// TIA Portal project "Project19" (V15.1)

(* hardware
DEVICE "S7-1200 station_1"  S7-1200 Station
   slot 0: "Rack_0"  S7-1200 Rack  Rack  V1.0
   slot 1: "PLC_1"  CPU 1214C DC/DC/DC  6ES7 214-1AG40-0XB0  V4.2
*)

// ===== PLC "PLC_1"  CPU 1214C DC/DC/DC =====

VAR_GLOBAL   // PLC tag table "Default tag table"
   "BE" AT %I0.0 : Bool;
   "LIGA" AT %I0.1 : Bool;
   "DESLIGA" AT %I0.2 : Bool;
   "SA0" AT %I0.3 : Bool;
   "SA1" AT %I0.4 : Bool;
   "SB0" AT %I0.5 : Bool;
   "SB1" AT %I0.6 : Bool;
   "SC0" AT %I0.7 : Bool;
   "SC1" AT %I1.0 : Bool;
   "SD0" AT %I1.1 : Bool;
   "SD1" AT %I1.2 : Bool;
   "AVANÇA A" AT %Q0.1 : Bool;
   "AVANÇA B" AT %Q0.2 : Bool;
   "AVANÇA C" AT %Q0.3 : Bool;
   "AVANÇA D" AT %Q0.4 : Bool;
   "RECUA A" AT %Q0.5 : Bool;
   "RECUA B" AT %Q0.6 : Bool;
   "RECUA C" AT %Q0.7 : Bool;
   "RECUA D" AT %Q1.0 : Bool;
   "LIGADA" AT %Q1.1 : Bool;
   "FALHA" AT %Q1.2 : Bool;
   "M1" AT %M0.0 : Bool;
   "M2" AT %M0.1 : Bool;
   "M3" AT %M0.2 : Bool;
   "M4" AT %M0.3 : Bool;
   "M5" AT %M0.4 : Bool;
   "M6" AT %M0.5 : Bool;
   "M7" AT %M0.6 : Bool;
END_VAR

DATA_BLOCK "CILINDRO_A_DB"   // DB1
{ S7_Optimized_Access := 'TRUE' }
VERSION : 0.1
// stored: InstanceOfName CILINDRO
"CILINDRO"
BEGIN
END_DATA_BLOCK

DATA_BLOCK "CILINDRO_B_DB"   // DB2
{ S7_Optimized_Access := 'TRUE' }
VERSION : 0.1
// stored: InstanceOfName CILINDRO
"CILINDRO"
BEGIN
END_DATA_BLOCK

DATA_BLOCK "CILINDRO_C_DB"   // DB5
{ S7_Optimized_Access := 'TRUE' }
VERSION : 0.1
// stored: InstanceOfName CILINDRO
"CILINDRO"
BEGIN
END_DATA_BLOCK

DATA_BLOCK "CILINDRO_D_DB"   // DB7
{ S7_Optimized_Access := 'TRUE' }
VERSION : 0.1
// stored: InstanceOfName CILINDRO
"CILINDRO"
BEGIN
END_DATA_BLOCK

// folder: System blocks/Program resources

DATA_BLOCK "T1"   // DB3
{ S7_Optimized_Access := 'TRUE' }
AUTHOR : Simatic
FAMILY : IEC
NAME : IEC_TMR
VERSION : 1.0
// stored: InstanceOfName IEC_TIMER
"IEC_TIMER"
BEGIN
END_DATA_BLOCK

DATA_BLOCK "T2"   // DB4
{ S7_Optimized_Access := 'TRUE' }
AUTHOR : Simatic
FAMILY : IEC
NAME : IEC_TMR
VERSION : 1.0
// stored: InstanceOfName IEC_TIMER
"IEC_TIMER"
BEGIN
END_DATA_BLOCK

DATA_BLOCK "T3"   // DB6
{ S7_Optimized_Access := 'TRUE' }
AUTHOR : Simatic
FAMILY : IEC
NAME : IEC_TMR
VERSION : 1.0
// stored: InstanceOfName IEC_TIMER
"IEC_TIMER"
BEGIN
END_DATA_BLOCK

DATA_BLOCK "T4"   // DB8
{ S7_Optimized_Access := 'TRUE' }
AUTHOR : Simatic
FAMILY : IEC
NAME : IEC_TMR
VERSION : 1.0
// stored: InstanceOfName IEC_TIMER
"IEC_TIMER"
BEGIN
END_DATA_BLOCK

// folder: (top level)

FUNCTION_BLOCK "CILINDRO"   // FB1, LAD
{ S7_Optimized_Access := 'TRUE' }
VERSION : 0.1
   VAR_INPUT
      "COMANDO AVANÇO" : Bool;
      "COMANDO RECUO" : Bool;
      "SENSOR AVANÇO" : Bool;
      "SENSOR RECUO" : Bool;
   END_VAR
   VAR_OUTPUT
      AVANÇO : Bool;
      RECUO : Bool;
   END_VAR
BEGIN

REGION Network 1
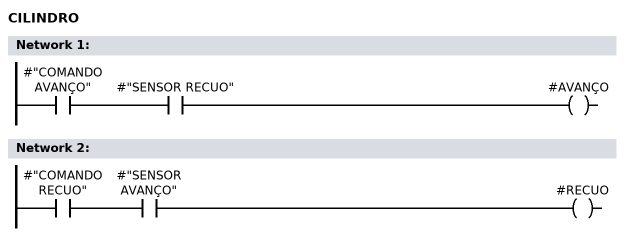
   RUNG wire#powerrail
      Contact( #"COMANDO AVANÇO" )
      Contact( #"SENSOR RECUO" )
      Coil( #AVANÇO )
   END_RUNG
   // the same network as SCL:
   #AVANÇO := #"COMANDO AVANÇO" AND #"SENSOR RECUO";
END_REGION

REGION Network 2
   RUNG wire#powerrail
      Contact( #"COMANDO RECUO" )
      Contact( #"SENSOR AVANÇO" )
      Coil( #RECUO )
   END_RUNG
   // the same network as SCL:
   #RECUO := #"COMANDO RECUO" AND #"SENSOR AVANÇO";
END_REGION
END_FUNCTION_BLOCK

FUNCTION "LOGICA DE ACIONAMENTO" : Void   // FC1, LAD
TITLE = Sequência dos cilindros
{ S7_Optimized_Access := 'TRUE' }
VERSION : 0.1
// A+B+5sA-5sB-C+5sD+5s(C-D-)
BEGIN

REGION Network 1: Selo ligado com memoria
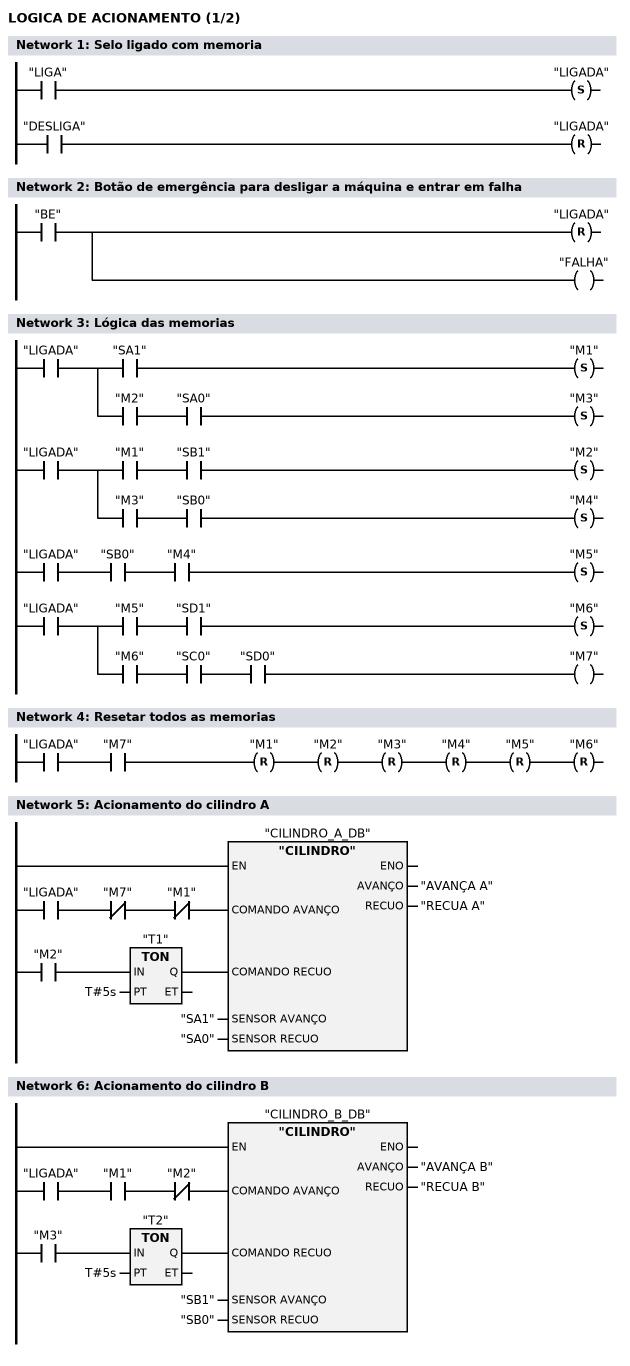
   RUNG wire#powerrail
      Contact( "LIGA" )
      S_Coil( "LIGADA" )
   END_RUNG
   RUNG wire#powerrail
      Contact( "DESLIGA" )
      R_Coil( "LIGADA" )
   END_RUNG
   // the same network as SCL:
   IF "LIGA" THEN "LIGADA" := TRUE; END_IF;
   IF "DESLIGA" THEN "LIGADA" := FALSE; END_IF;
END_REGION

REGION Network 2: Botão de emergência para desligar a máquina e entrar em falha
   RUNG wire#powerrail
      Contact( "BE" )
      wire#w1
      R_Coil( "LIGADA" )
   END_RUNG
   RUNG wire#w1
      Coil( "FALHA" )
   END_RUNG
   // the same network as SCL:
   IF "BE" THEN "LIGADA" := FALSE; END_IF;
   "FALHA" := "BE";
END_REGION

REGION Network 3: Lógica das memorias
   RUNG wire#powerrail
      Contact( "LIGADA" )
      wire#w1
      Contact( "SA1" )
      S_Coil( "M1" )
   END_RUNG
   RUNG wire#w1
      Contact( "M2" )
      Contact( "SA0" )
      S_Coil( "M3" )
   END_RUNG
   RUNG wire#powerrail
      Contact( "LIGADA" )
      wire#w2
      Contact( "M1" )
      Contact( "SB1" )
      S_Coil( "M2" )
   END_RUNG
   RUNG wire#w2
      Contact( "M3" )
      Contact( "SB0" )
      S_Coil( "M4" )
   END_RUNG
   RUNG wire#powerrail
      Contact( "LIGADA" )
      Contact( "SB0" )
      Contact( "M4" )
      S_Coil( "M5" )
   END_RUNG
   RUNG wire#powerrail
      Contact( "LIGADA" )
      wire#w3
      Contact( "M5" )
      Contact( "SD1" )
      S_Coil( "M6" )
   END_RUNG
   RUNG wire#w3
      Contact( "M6" )
      Contact( "SC0" )
      Contact( "SD0" )
      Coil( "M7" )
   END_RUNG
   // the same network as SCL:
   IF "LIGADA" AND "SA1" THEN "M1" := TRUE; END_IF;
   IF "LIGADA" AND "M2" AND "SA0" THEN "M3" := TRUE; END_IF;
   IF "LIGADA" AND "M1" AND "SB1" THEN "M2" := TRUE; END_IF;
   IF "LIGADA" AND "M3" AND "SB0" THEN "M4" := TRUE; END_IF;
   IF "LIGADA" AND "SB0" AND "M4" THEN "M5" := TRUE; END_IF;
   IF "LIGADA" AND "M5" AND "SD1" THEN "M6" := TRUE; END_IF;
   "M7" := "LIGADA" AND "M6" AND "SC0" AND "SD0";
END_REGION

REGION Network 4: Resetar todos as memorias
   RUNG wire#powerrail
      Contact( "LIGADA" )
      Contact( "M7" )
      R_Coil( "M1" )
      R_Coil( "M2" )
      R_Coil( "M3" )
      R_Coil( "M4" )
      R_Coil( "M5" )
      R_Coil( "M6" )
   END_RUNG
   // the same network as SCL:
   IF "LIGADA" AND "M7" THEN
       "M1" := FALSE;
       "M2" := FALSE;
       "M3" := FALSE;
       "M4" := FALSE;
       "M5" := FALSE;
       "M6" := FALSE;
   END_IF;
END_REGION

REGION Network 5: Acionamento do cilindro A
   "T1".TON(IN := "M2", PT := T#5s);
   "CILINDRO_A_DB"("COMANDO AVANÇO" := "LIGADA" AND NOT "M7" AND NOT "M1",   // "CILINDRO"
                   "COMANDO RECUO" := "T1".Q,
                   "SENSOR AVANÇO" := "SA1",
                   "SENSOR RECUO" := "SA0",
                   AVANÇO => "AVANÇA A",
                   RECUO => "RECUA A");
END_REGION

REGION Network 6: Acionamento do cilindro B
   "T2".TON(IN := "M3", PT := T#5s);
   "CILINDRO_B_DB"("COMANDO AVANÇO" := "LIGADA" AND "M1" AND NOT "M2",   // "CILINDRO"
                   "COMANDO RECUO" := "T2".Q,
                   "SENSOR AVANÇO" := "SB1",
                   "SENSOR RECUO" := "SB0",
                   AVANÇO => "AVANÇA B",
                   RECUO => "RECUA B");
END_REGION

REGION Network 7: Acionamento do cilindro C
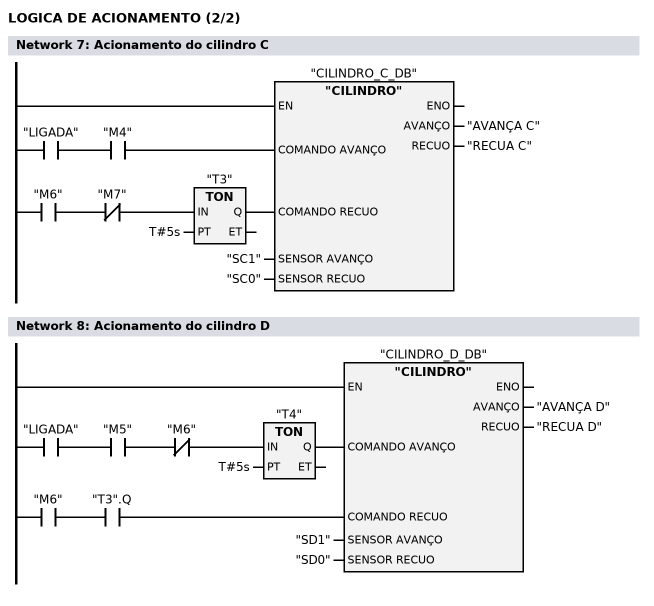
   "T3".TON(IN := "M6" AND NOT "M7", PT := T#5s);
   "CILINDRO_C_DB"("COMANDO AVANÇO" := "LIGADA" AND "M4",   // "CILINDRO"
                   "COMANDO RECUO" := "T3".Q,
                   "SENSOR AVANÇO" := "SC1",
                   "SENSOR RECUO" := "SC0",
                   AVANÇO => "AVANÇA C",
                   RECUO => "RECUA C");
END_REGION

REGION Network 8: Acionamento do cilindro D
   "T4".TON(IN := "LIGADA" AND "M5" AND NOT "M6", PT := T#5s);
   "CILINDRO_D_DB"("COMANDO AVANÇO" := "T4".Q,   // "CILINDRO"
                   "COMANDO RECUO" := "M6" AND "T3".Q,
                   "SENSOR AVANÇO" := "SD1",
                   "SENSOR RECUO" := "SD0",
                   AVANÇO => "AVANÇA D",
                   RECUO => "RECUA D");
END_REGION
END_FUNCTION

ORGANIZATION_BLOCK "Main"   // OB1, LAD, ProgramCycle
TITLE = "Main Program Sweep (Cycle)"
{ S7_Optimized_Access := 'TRUE' }
VERSION : 0.1
   VAR_INPUT
      Initial_Call : Bool;   // Initial call of this OB
      Remanence : Bool;   // =True, if remanent data are available
   END_VAR
BEGIN

REGION Network 1
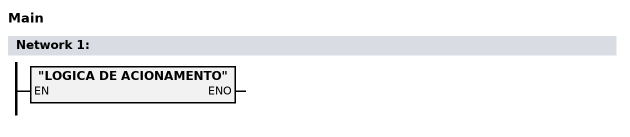
   RUNG wire#powerrail
      "LOGICA DE ACIONAMENTO"()
   END_RUNG
   // the same network as SCL:
   "LOGICA DE ACIONAMENTO"();
END_REGION
END_ORGANIZATION_BLOCK